(* IEC 61131-3 sources: Lasal/CPU_5344_V01/Class/andServerClient, 1 file *)

(* ---- andServerClient.st ---- *)
(*!
<Class
	Name               = "andServerClient"
	Revision           = "0.0"
	RealtimeTask       = "false"
	CyclicTask         = "false"
	BackgroundTask     = "false"
	Sigmatek           = "false"
	OSInterface        = "false"
	HighPriority       = "false"
	Automatic          = "false"
	UpdateMode         = "Prescan"
	SharedCommandTable = "true"
	Objectsize         = "(284,120)">
	<Channels>
		<Server Name="ClassSvr" Visualized="false" Initialize="false" WriteProtected="false" Retentive="false"/>
		<Client Name="client1" Required="true" Internal="false"/>
		<Client Name="client2" Required="true" Internal="false"/>
		<Client Name="client3" Required="false" Internal="false"/>
		<Client Name="client4" Required="false" Internal="false"/>
	</Channels>
</Class>
*)
andServerClient : CLASS
  //Servers:
	ClassSvr 	: SvrChCmd_DINT;
  //Clients:
	client1 	: CltCh_DINT;
	client2 	: CltCh_DINT;
	client3 	: CltCh_DINT;
	client4 	: CltCh_DINT;
  //Variables:
  //Functions:

	FUNCTION VIRTUAL GLOBAL ClassSvr::Write
		VAR_INPUT
			input (EAX) 	: DINT;
		END_VAR
		VAR_OUTPUT
			result (EAX) 	: DINT;
		END_VAR;
  //Tables:
	FUNCTION @STD
		VAR_OUTPUT
			ret_code	: CONFSTATES;
		END_VAR;
	FUNCTION GLOBAL TAB @CT_;
END_CLASS;

// JdK 22-7-2019: andServerClient created for Traffiroad/4284

// goal is to write server to 4 clients

FUNCTION VIRTUAL GLOBAL andServerClient::ClassSvr::Write
	VAR_INPUT
		input (EAX) 	: DINT;
	END_VAR
	VAR_OUTPUT
		result (EAX) 	: DINT;
	END_VAR

	ClassSvr := input;
  client1:= ClassSvr;
  client2:= ClassSvr;
  client3:= ClassSvr;
  client4:= ClassSvr;
  client1.Write(input:=client1);
  client2.Write(input:=client2);
  client3.Write(input:=client3);
  client4.Write(input:=client4);
	result := ClassSvr;

END_FUNCTION
